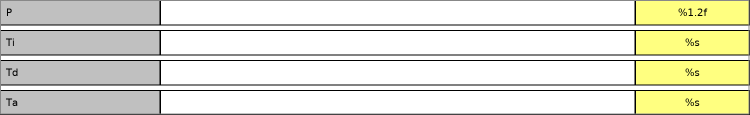
VISUALIZATION VISU_CONFIG_EFF  // 750x115
VAR_IN_OUT
	m_Input_PRG_EFFLUVAGE : BLOCK_PRG_EFFLUVAGE;
END_VAR
    Rectangle (160,0 475x25), text list: 'TextList_Config_EFFLUVAGE', text index: 4
    Rectangle (635,0 115x25), "%1.2f", text variable: m_Input_PRG_EFFLUVAGE.Effluvage.ALEFF.CONF_Kp, input disabled if: NOT Global_Variables.PRG_USER.ACTU_USER.CONF_MACHINE
        OnMouseClick: write the text variable via InputWithLimits, min 0
    Rectangle (0,0 160x25), "P"
    Rectangle (160,30 475x25), text list: 'TextList_Config_EFFLUVAGE', text index: 5
    Rectangle (635,30 115x25), "%s", text variable: m_Input_PRG_EFFLUVAGE.Effluvage.ALEFF.CONF_Tn, input disabled if: NOT Global_Variables.PRG_USER.ACTU_USER.CONF_MACHINE
        OnMouseClick: write the text variable via InputWithLimits
    Rectangle (0,30 160x25), "Ti"
    Rectangle (0,60 160x25), "Td"
    Rectangle (160,60 475x25), text list: 'TextList_Config_EFFLUVAGE', text index: 6
    Rectangle (635,60 115x25), "%s", text variable: m_Input_PRG_EFFLUVAGE.Effluvage.ALEFF.CONF_Tv, input disabled if: NOT Global_Variables.PRG_USER.ACTU_USER.CONF_MACHINE
        OnMouseClick: write the text variable via InputWithLimits
    Rectangle (0,90 160x25), "Ta"
    Rectangle (160,90 475x25), text list: 'TextList_Config_EFFLUVAGE', text index: 7
    Rectangle (635,90 115x25), "%s", text variable: m_Input_PRG_EFFLUVAGE.Effluvage.ALEFF.CONF_Td, input disabled if: NOT Global_Variables.PRG_USER.ACTU_USER.CONF_MACHINE
        OnMouseClick: write the text variable via InputWithLimits
END_VISUALIZATION

(* stored: Version 1.1.0.1, ProductVersion 3.1.4024.10
   Visu VISU_CONFIG_EFF: Id {c1052857-3f4b-4b6b-8a5d-0faa7377438e} *)
